{attribute 'qualified_only'}
VAR_GLOBAL
END_VAR

(* stored: Version 1.1.0.1, ProductVersion 3.1.4024.12
   GVL G_Task2: Id {734fe8fc-1960-4684-8004-5362632b17d1} *)
